// TIA Portal V17 export
// export: Created 2025-03-07T09:23:46.8910198Z, ExportSetting WithDefaults, DisplayName Totally Integrated Automation Portal, DisplayVersion V17 Update 8, DisplayName TIA Portal Openness, DisplayVersion V17 Update 8, DisplayName TIA Portal Version Control Interface, DisplayVersion V17, DisplayName SINAMICS Startdrive Advanced, DisplayVersion V17 SP2, DisplayName SINAMICS Startdrive G110M, G120, G120C, G120D, G120P, G115D, DisplayVersion V17 SP2, DisplayName SINAMICS Startdrive G130, G150, S120, S150, SINAMICS MV, S210, DisplayVersion V17 SP2, DisplayName STEP 7 Professional, DisplayVersion V17 Update 8, DisplayName SINUMERIK ONE STEP 7 Toolbox, DisplayVersion V17 Update 12, DisplayName SINUMERIK 840D sl STEP 7 Toolbox, DisplayVersion V17 Update 12, DisplayName STEP 7 Safety, DisplayVersion V17 Update 6, DisplayName WinCC Advanced, DisplayVersion V17 Update 8
DATA_BLOCK "DB7270_HOPPER_1_UNIT_01"   // DB7270
{ DB_Accessible_From_OPC_UA := 'FALSE' }
VERSION : 0.1
// stored: AutoNumber false, DBAccessibleFromOPCUA false, DBAccessibleFromWebserver true, InstanceOfName FB7240_VARIABLES_PLC_HMI_HOPPERS, InstanceOfType FB
"FB7240_VARIABLES_PLC_HMI_HOPPERS"
   // VAR_INPUT
   //    STIRRER_SPEED_ACTUAL : DInt;
   //    STIRRER_SPEED_CONS : DInt;
   //    UPPER_JACKET_ACTUAL : Real;
   //    UPPER_JACKET_CONS : Real;
   //    LOWER_JACKET_ACTUAL : Real;
   //    LOWER_JACKET_CONS : Real;
   //    HOPPER_COVER_ACTUAL : Real;
   //    HOPPER_COVER_CONS : Real;
   //    FEEDING_COVER_ACTUAL : Real;
   //    FEEDER_DISK_PRESS_ACTUAL : Real;
   //    MAX_WEIGHT_ACTUAL : Real;
   //    TOTAL_WEIGHT_ACTUAL : Real;
   //    HOPPER_WEIGHT_ACTUAL : Real;
   //    POWDER_WEIGHT_ACTUAL : Real;
   // END_VAR
   // VAR_OUTPUT
   //    STIRRER_SPEED_SETPOINT : DInt;
   //    UPPER_JACKET_SETPOINT : Real;
   //    LOWER_JACKET_SETPOINT : Real;
   //    HOPPER_COVER_SETPOINT : Real;
   //    HOPPER_WEIGHT_INPUT : Real;
   //    MAX_WEIGHT_INPUT : Real;
   // END_VAR
   // VAR_IN_OUT
   //    HOPPER_LINE_IN_OUT : "UDT_Hopper Line";
   // END_VAR
BEGIN
END_DATA_BLOCK
